(* PLC project MotorControlTemplate, Industrial AI Agent CODESYS 3.5.21.0 *)
(* stored: creationDateTime 2026-06-10T10:00:00, modificationDateTime 2026-06-10T10:00:00 *)

FUNCTION_BLOCK FB_MotorControl
  VAR_INPUT
    xStart : BOOL;  (* Calistirma komutu (start) *)
    xStop : BOOL;  (* Durdurma komutu (stop, oncelikli) *)
    xInterlock : BOOL;  (* Guvenlik kilidi: TRUE = calismaya izin var *)
  END_VAR
  VAR_OUTPUT
    xRun : BOOL;  (* Motor calisma cikisi *)
    xFault : BOOL;  (* Hata bayragi (interlock kayboldu) *)
  END_VAR
  VAR
    fbRS : RS;
  END_VAR

                        
// ------------------------------------------------------------
// FB_MotorControl - Mandalli (RS) motor kontrol blogu
// Stop ve interlock kaybi oncelikli olarak motoru durdurur.
// RS flip-flop: Set = xStart, Reset (oncelikli) = stop kosulu
// ------------------------------------------------------------

// Interlock kaybi hata uretir
xFault := NOT xInterlock;

// RS mandali: Set1 baskin reset, R baskin
fbRS(
    SET  := xStart AND xInterlock,
    RESET1 := xStop OR NOT xInterlock
);

xRun := fbRS.Q1;

                    
END_FUNCTION_BLOCK
